// Mitsubishi GX Works2 project: Lab_3_insys_P_J   PLC: FX1N/FX1NC

// global labels: Global1
VAR_GLOBAL
  stopp AT X000 : BOOL;
  start AT X001 : BOOL;
  motorvern AT X002 : BOOL;
  endebryter_A_fremme2 AT X003 : BOOL;
  endebryter_A_tilbake2 AT X004 : BOOL;
  endebryter_Bor_nede AT X006 : BOOL;
  endebryter_Bor_oppe AT X005 : BOOL;
  endebryter_C_fremme2 AT X007 : BOOL;
  endebryter_C_tilbake2 AT X010 : BOOL;
  kontaktor_K1 AT Y000 : BOOL;
  A_frem AT Y001 : BOOL;
  A_tilbake AT Y002 : BOOL;
  Bor_opp AT Y003 : BOOL;
  Bor_ned AT Y004 : BOOL;
  C_frem AT Y005 : BOOL;
  C_tilbake AT Y006 : BOOL;
END_VAR

// task Task_01 (event TRUE, interval 0, priority 31): borelabb

PROGRAM borelabb
(* structured ladder/FBD written out as ST: instructions are called as NAME(EN, inputs, outputs); _pN, _eN, _tN stand for wires *)
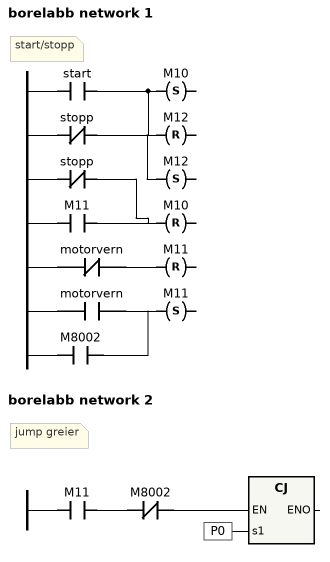
(* network 1 *)
(* start/stopp *)
SET(start, M10);
RST(start, M12);
SET(NOT stopp, M12);
RST((NOT stopp) OR M11, M10);
RST(NOT motorvern, M11);
SET(motorvern OR M8002, M11);
(* network 2 *)
(* jump greier *)
CJ(M11 AND NOT M8002, P0);
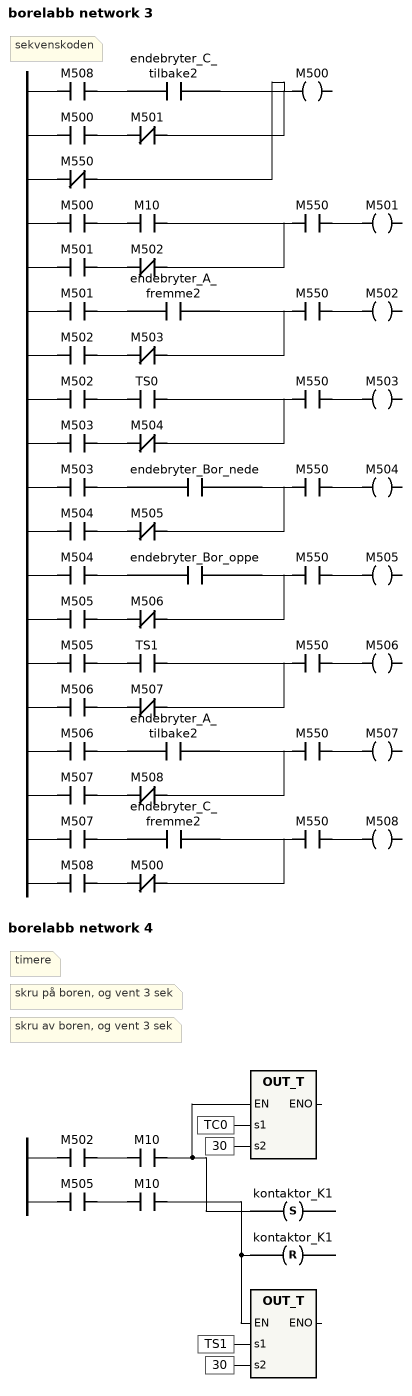
(* network 3 *)
(* sekvenskoden *)
M500 := (M508 AND endebryter_C_tilbake2) OR (M500 AND NOT M501) OR (NOT M550);
M501 := ((M500 AND M10) OR (M501 AND NOT M502)) AND M550;
M502 := ((M501 AND endebryter_A_fremme2) OR (M502 AND NOT M503)) AND M550;
M503 := ((M502 AND TS0) OR (M503 AND NOT M504)) AND M550;
M504 := ((M503 AND endebryter_Bor_nede) OR (M504 AND NOT M505)) AND M550;
M505 := ((M504 AND endebryter_Bor_oppe) OR (M505 AND NOT M506)) AND M550;
M506 := ((M505 AND TS1) OR (M506 AND NOT M507)) AND M550;
M507 := ((M506 AND endebryter_A_tilbake2) OR (M507 AND NOT M508)) AND M550;
M508 := ((M507 AND endebryter_C_fremme2) OR (M508 AND NOT M500)) AND M550;
(* network 4 P0: P0 *)
(* timere *)
(* skru på boren, og vent 3 sek *)
(* skru av boren, og vent 3 sek *)
_p1 := M502 AND M10;
SET(_p1, kontaktor_K1);
OUT_T(_p1, TC0, 30);
_p2 := M505 AND M10;
RST(_p2, kontaktor_K1);
OUT_T(_p2, TS1, 30);
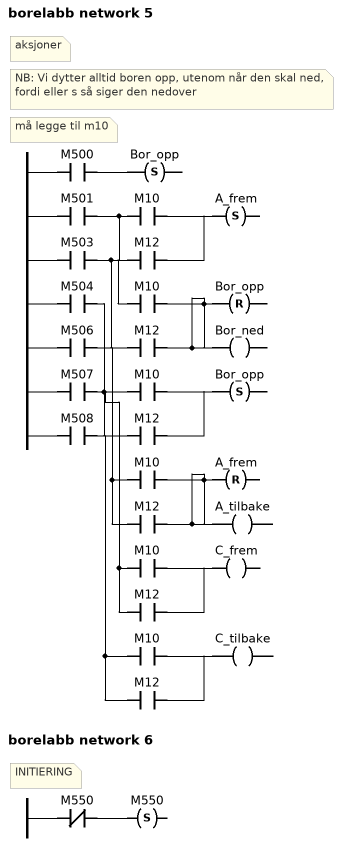
(* network 5 *)
(* aksjoner *)
(* NB: Vi dytter alltid boren opp, utenom når den skal ned, fordi eller s så siger den nedover *)
(* må legge til m10 *)
SET(M500, Bor_opp);
SET((M501 AND M10) OR (M501 AND M12), A_frem);
_p1 := (M503 AND M10) OR (M503 AND M12);
RST(_p1, Bor_opp);
Bor_ned := _p1;
SET((M504 AND M10) OR (M504 AND M12), Bor_opp);
_p2 := (M506 AND M10) OR (M506 AND M12);
RST(_p2, A_frem);
A_tilbake := _p2;
C_frem := (M507 AND M10) OR (M507 AND M12);
C_tilbake := (M508 AND M10) OR (M508 AND M12);
(* network 6 *)
(* INITIERING *)
SET(NOT M550, M550);
END_PROGRAM
